FUNCTION_BLOCK FB_System_AFA_Ablaufsteuerung
VAR_IN_OUT
	Zustand					: ST_System_AFA_Zustand;
	Stellwert				: ST_System_AFA_Stellwert;
	Steuerung				: ST_System_AFA_Steuerung;
END_VAR
VAR_INPUT
	Zustand_Stellventil		: ST_SVs_Zustand;
	Zustand_Pumpe			: ST_PU_Zustand;
	Zustand_Regelventil		: ST_RV_Zustand;
END_VAR
VAR_OUTPUT
END_VAR
VAR
END_VAR

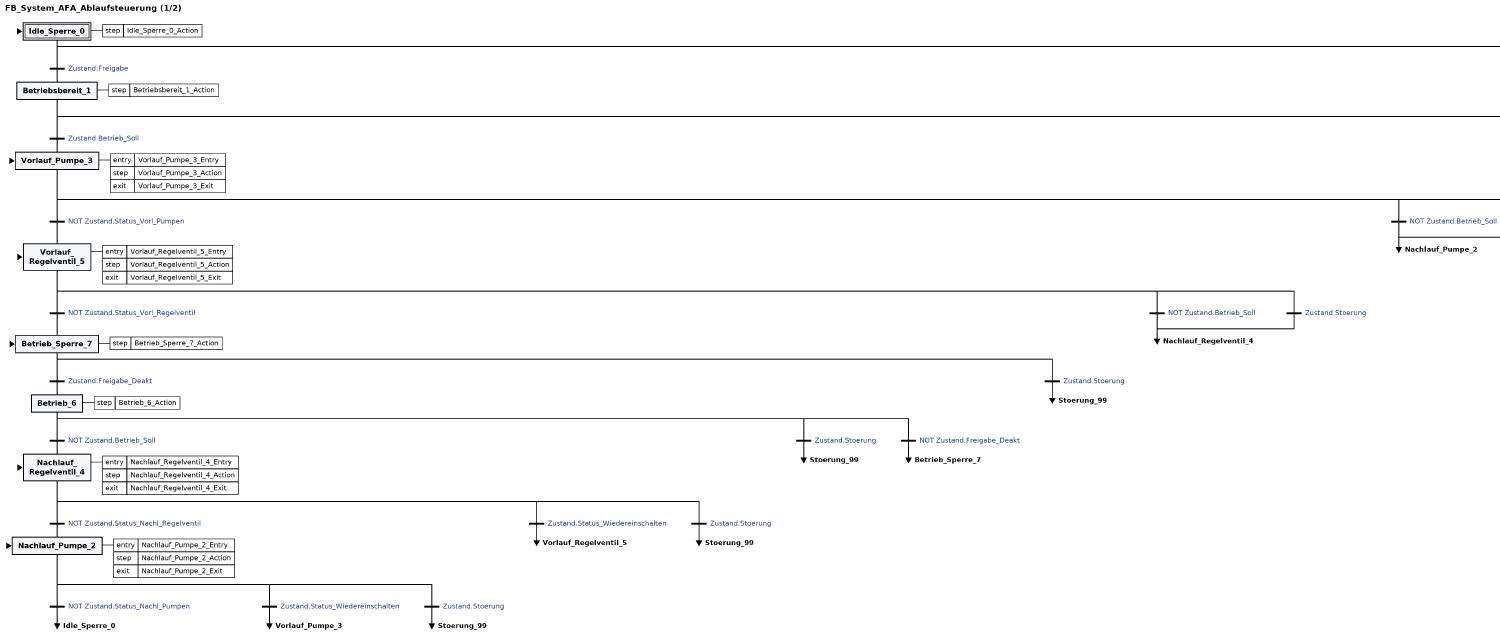
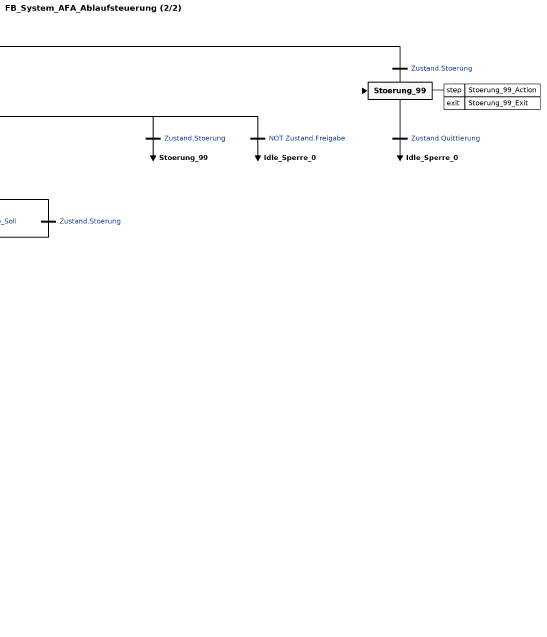
INITIAL_STEP Idle_Sperre_0:
    Idle_Sperre_0_Action(N);  // step action
END_STEP
TRANSITION FROM Idle_Sperre_0 TO Betriebsbereit_1
    := Zustand.Freigabe;
END_TRANSITION
TRANSITION FROM Idle_Sperre_0 TO Stoerung_99
    := Zustand.Stoerung;
END_TRANSITION
STEP Stoerung_99:
    Stoerung_99_Action(N);  // step action
    Stoerung_99_Exit(P0);  // exit action
END_STEP
TRANSITION FROM Stoerung_99 TO Idle_Sperre_0
    := Zustand.Quittierung;
END_TRANSITION
STEP Betriebsbereit_1:
    Betriebsbereit_1_Action(N);  // step action
END_STEP
TRANSITION FROM Betriebsbereit_1 TO Vorlauf_Pumpe_3
    := Zustand.Betrieb_Soll;
END_TRANSITION
TRANSITION FROM Betriebsbereit_1 TO Stoerung_99
    := Zustand.Stoerung;
END_TRANSITION
TRANSITION FROM Betriebsbereit_1 TO Idle_Sperre_0
    := NOT Zustand.Freigabe;
END_TRANSITION
STEP Vorlauf_Pumpe_3:
    Vorlauf_Pumpe_3_Entry(P1);  // entry action
    Vorlauf_Pumpe_3_Action(N);  // step action
    Vorlauf_Pumpe_3_Exit(P0);  // exit action
END_STEP
TRANSITION FROM Vorlauf_Pumpe_3 TO Vorlauf_Regelventil_5
    := NOT Zustand.Status_Vorl_Pumpen;
END_TRANSITION
TRANSITION FROM Vorlauf_Pumpe_3 TO Nachlauf_Pumpe_2
    := NOT Zustand.Betrieb_Soll;
END_TRANSITION
TRANSITION FROM Vorlauf_Pumpe_3 TO Nachlauf_Pumpe_2
    := Zustand.Stoerung;
END_TRANSITION
STEP Vorlauf_Regelventil_5:
    Vorlauf_Regelventil_5_Entry(P1);  // entry action
    Vorlauf_Regelventil_5_Action(N);  // step action
    Vorlauf_Regelventil_5_Exit(P0);  // exit action
END_STEP
TRANSITION FROM Vorlauf_Regelventil_5 TO Betrieb_Sperre_7
    := NOT Zustand.Status_Vorl_Regelventil;
END_TRANSITION
TRANSITION FROM Vorlauf_Regelventil_5 TO Nachlauf_Regelventil_4
    := NOT Zustand.Betrieb_Soll;
END_TRANSITION
TRANSITION FROM Vorlauf_Regelventil_5 TO Nachlauf_Regelventil_4
    := Zustand.Stoerung;
END_TRANSITION
STEP Betrieb_Sperre_7:
    Betrieb_Sperre_7_Action(N);  // step action
END_STEP
TRANSITION FROM Betrieb_Sperre_7 TO Betrieb_6
    := Zustand.Freigabe_Deakt;
END_TRANSITION
TRANSITION FROM Betrieb_Sperre_7 TO Stoerung_99
    := Zustand.Stoerung;
END_TRANSITION
STEP Betrieb_6:
    Betrieb_6_Action(N);  // step action
END_STEP
TRANSITION FROM Betrieb_6 TO Nachlauf_Regelventil_4
    := NOT Zustand.Betrieb_Soll;
END_TRANSITION
TRANSITION FROM Betrieb_6 TO Stoerung_99
    := Zustand.Stoerung;
END_TRANSITION
TRANSITION FROM Betrieb_6 TO Betrieb_Sperre_7
    := NOT Zustand.Freigabe_Deakt;
END_TRANSITION
STEP Nachlauf_Regelventil_4:
    Nachlauf_Regelventil_4_Entry(P1);  // entry action
    Nachlauf_Regelventil_4_Action(N);  // step action
    Nachlauf_Regelventil_4_Exit(P0);  // exit action
END_STEP
TRANSITION FROM Nachlauf_Regelventil_4 TO Nachlauf_Pumpe_2
    := NOT Zustand.Status_Nachl_Regelventil;
END_TRANSITION
TRANSITION FROM Nachlauf_Regelventil_4 TO Vorlauf_Regelventil_5
    := Zustand.Status_Wiedereinschalten;
END_TRANSITION
TRANSITION FROM Nachlauf_Regelventil_4 TO Stoerung_99
    := Zustand.Stoerung;
END_TRANSITION
STEP Nachlauf_Pumpe_2:
    Nachlauf_Pumpe_2_Entry(P1);  // entry action
    Nachlauf_Pumpe_2_Action(N);  // step action
    Nachlauf_Pumpe_2_Exit(P0);  // exit action
END_STEP
TRANSITION FROM Nachlauf_Pumpe_2 TO Idle_Sperre_0
    := NOT Zustand.Status_Nachl_Pumpen;
END_TRANSITION
TRANSITION FROM Nachlauf_Pumpe_2 TO Vorlauf_Pumpe_3
    := Zustand.Status_Wiedereinschalten;
END_TRANSITION
TRANSITION FROM Nachlauf_Pumpe_2 TO Stoerung_99
    := Zustand.Stoerung;
END_TRANSITION

ACTION Betrieb_6_Action:
(* Stellwert setzen *)
Stellwert.Anford_Pumpe		:= TRUE;
Stellwert.Anford_Regelventil		:= TRUE;

(* Zustand setzen *)
Zustand.Betrieb				:= TRUE;
Zustand.Status				:= E_System_AFA_Zustand_Status_Betrieb;
END_ACTION

ACTION Betrieb_Sperre_7_Action:
(* Stellwert setzen *)
Stellwert.Anford_Pumpe		:= TRUE;
Stellwert.Anford_Regelventil		:= TRUE;

(* Zustand setzen *)
Zustand.Betrieb				:= TRUE;
Zustand.Status				:= E_System_AFA_Zustand_Status_Betrieb_Sperre;
END_ACTION

ACTION Betriebsbereit_1_Action:
(* Stellwert setzen *)
Stellwert.Anford_Pumpe	:= FALSE;
Stellwert.Anford_Regelventil	:= FALSE;

(* Zustand setzen *)
Zustand.Betrieb			:= FALSE;
Zustand.Status			:= E_System_AFA_Zustand_Status_Betriebsbereit;
END_ACTION

ACTION Idle_Sperre_0_Action:
(* Stellwert setzen *)
Stellwert.Anford_Pumpe	:= FALSE;
Stellwert.Anford_Regelventil	:= FALSE;

(* Zustand setzen *)
Zustand.Betrieb			:= FALSE;
Zustand.Status			:= E_System_AFA_Zustand_Status_Idle_Sperre;


(* Quittierungszustand auf False setzen, damit das System bei einer erneuten Störung nicht direkt wieder angeschaltet wird *)
Steuerung.Quittierung	:= FALSE;
END_ACTION

ACTION Nachlauf_Pumpe_2_Action:
(* Stellwert setzen *)
Stellwert.Anford_Pumpe		:= FALSE;
Stellwert.Anford_Regelventil		:= FALSE;

(* Zustand setzen *)
Zustand.Betrieb				:= FALSE;
Zustand.Status				:= E_System_AFA_Zustand_Status_Nachl_Pumpe;
Zustand.Status_Nachl_Pumpen	:= Zustand_Pumpe.Betrieb OR Zustand_Pumpe.Status_Nachl;
Zustand.Status_Wiedereinschalten := Zustand.Betrieb_Soll AND Stellwert.Einschalten;
END_ACTION

ACTION Nachlauf_Pumpe_2_Entry:
Zustand.Status_Nachl_Pumpen	:= TRUE;
END_ACTION

ACTION Nachlauf_Pumpe_2_Exit:
Zustand.Status_Nachl_Pumpen	:= FALSE;
END_ACTION

ACTION Nachlauf_Regelventil_4_Action:
(* Stellwert setzen *)
Stellwert.Anford_Pumpe		:= TRUE;
Stellwert.Anford_Regelventil		:= FALSE;

(* Zustand setzen *)
Zustand.Betrieb					:= FALSE;
Zustand.Status					:= E_System_AFA_Zustand_Status_Nachl_Regelventil;
Zustand.Status_Nachl_Regelventil	:= Zustand_Regelventil.Betrieb OR Zustand_Regelventil.Status_Nachl;
Zustand.Status_Wiedereinschalten := Zustand.Betrieb_Soll AND Stellwert.Einschalten;
END_ACTION

ACTION Nachlauf_Regelventil_4_Entry:
Zustand.Status_Nachl_Regelventil		:= TRUE;
END_ACTION

ACTION Nachlauf_Regelventil_4_Exit:
Zustand.Status_Nachl_Regelventil		:= FALSE;
END_ACTION

ACTION Stoerung_99_Action:
(* Stellwert setzen *)
Stellwert.Anford_Pumpe			:= FALSE;
Stellwert.Anford_Regelventil	:= FALSE;

(* Zustand setzen *)
Zustand.Betrieb					:= FALSE;
Zustand.Stoerung				:= TRUE;
Zustand.Status					:= E_System_AFA_Zustand_Status_Stoerung;
END_ACTION

ACTION Stoerung_99_Exit:
Zustand.Stoerung	:= FALSE;
END_ACTION

ACTION Vorlauf_Pumpe_3_Action:
(* Stellwert setzen *)
Stellwert.Anford_Pumpe		:= TRUE;
Stellwert.Anford_Regelventil		:= FALSE;

(* Zustand setzen *)
Zustand.Betrieb				:= FALSE;
Zustand.Status				:= E_System_AFA_Zustand_Status_Vorl_Pumpe;
Zustand.Status_Vorl_Pumpen	:= NOT(Zustand_Pumpe.Betrieb AND NOT Zustand_Pumpe.Status_Vorl);
END_ACTION

ACTION Vorlauf_Pumpe_3_Entry:
Zustand.Status_Vorl_Pumpen	:= TRUE;
END_ACTION

ACTION Vorlauf_Pumpe_3_Exit:
Zustand.Status_Vorl_Pumpen	:= FALSE;
END_ACTION

ACTION Vorlauf_Regelventil_5_Action:
(* Stellwert setzen *)
Stellwert.Anford_Pumpe		:= TRUE;
Stellwert.Anford_Regelventil		:= TRUE;

(* Zustand setzen *)
Zustand.Betrieb				:= FALSE;
Zustand.Status				:= E_System_AFA_Zustand_Status_Vorl_Regelventil;
Zustand.Status_Vorl_Regelventil	:= NOT(Zustand_Regelventil.Betrieb AND NOT Zustand_Regelventil.Status_Vorl);
END_ACTION

ACTION Vorlauf_Regelventil_5_Entry:
Zustand.Status_Vorl_Regelventil	:= TRUE;
END_ACTION

ACTION Vorlauf_Regelventil_5_Exit:
Zustand.Status_Vorl_Regelventil		:= FALSE;
END_ACTION

END_FUNCTION_BLOCK

(* stored: Version 1.1.0.1, ProductVersion 3.1.4024.9
   POU FB_System_AFA_Ablaufsteuerung: Id {6eb9e7a5-4bcf-4fdd-ba20-121b996afe54}, SpecialFunc None
   Action Betrieb_6_Action: Id {cd7393bd-be22-4f4e-80f6-729d5b239252}
   Action Betrieb_Sperre_7_Action: Id {9aeb56d1-63c7-468a-b58d-ab3b098e3a90}
   Action Betriebsbereit_1_Action: Id {bca28ff7-9051-441a-a293-3fe8f096bf39}
   Action Idle_Sperre_0_Action: Id {764a8c38-a66a-43a1-9878-80dd4a920c9e}
   Action Nachlauf_Pumpe_2_Action: Id {b13b8c66-c320-4341-a2bf-6d41b738ac46}
   Action Nachlauf_Pumpe_2_Entry: Id {d9123625-0355-4474-92a5-81b90cdf2ce9}
   Action Nachlauf_Pumpe_2_Exit: Id {304438c2-525c-4ed9-8092-baca78e3bc64}
   Action Nachlauf_Regelventil_4_Action: Id {2521c718-c609-47d4-9a23-07dcbb23873c}
   Action Nachlauf_Regelventil_4_Entry: Id {67195eb0-0081-470b-87c0-f3853015834a}
   Action Nachlauf_Regelventil_4_Exit: Id {3a3c3135-551c-4c92-8980-7a2b3688fe8a}
   Action Stoerung_99_Action: Id {e25d9b0a-8277-4b9b-a6bb-bae873450429}
   Action Stoerung_99_Exit: Id {144454ad-a3fe-4628-8cb8-119328ed914b}
   Action Vorlauf_Pumpe_3_Action: Id {822ebd89-9ee1-4fa3-966d-ae6e01237a3a}
   Action Vorlauf_Pumpe_3_Entry: Id {7bd96829-13a3-4408-9678-e76ef6fd613e}
   Action Vorlauf_Pumpe_3_Exit: Id {2ca2b164-abfd-45d9-9024-8892e02873f9}
   Action Vorlauf_Regelventil_5_Action: Id {471bea80-6870-475e-8e14-cd9054d2c8ca}
   Action Vorlauf_Regelventil_5_Entry: Id {617f39f0-c40b-48e4-b58d-024f943faa5f}
   Action Vorlauf_Regelventil_5_Exit: Id {b793e6e0-e63b-476e-b3bc-f593960f747a} *)
